{attribute 'GeneratedUsingTerminal: EL6201-0000-0017'}
{attribute addProperty BoxType "EL6201-0000-0017"}
{attribute addProperty Id "Slave_20A_DO0BOOL1Slave_20A_DO1BOOL1Slave_20A_DO2BOOL1Slave_20A_DO3BOOL1Slave_20B_DO0BOOL1Slave_20B_DO1BOOL1Slave_20B_DO2BOOL1Slave_20B_DO3BOOL1"}
{attribute addProperty CRC "2580098861"}
{attribute addProperty Size "8"}
TYPE Slave_20_Outputs_99C92F2D :
STRUCT
	{attribute addProperty Name "Slave_20A_DO0"}
	Slave_20A_DO0 : BOOL;
	{attribute addProperty Name "Slave_20A_DO1"}
	Slave_20A_DO1 : BOOL;
	{attribute addProperty Name "Slave_20A_DO2"}
	Slave_20A_DO2 : BOOL;
	{attribute addProperty Name "Slave_20A_DO3"}
	Slave_20A_DO3 : BOOL;
	{attribute addProperty Name "Slave_20B_DO0"}
	Slave_20B_DO0 : BOOL;
	{attribute addProperty Name "Slave_20B_DO1"}
	Slave_20B_DO1 : BOOL;
	{attribute addProperty Name "Slave_20B_DO2"}
	Slave_20B_DO2 : BOOL;
	{attribute addProperty Name "Slave_20B_DO3"}
	Slave_20B_DO3 : BOOL;
END_STRUCT
END_TYPE

(* stored: Version 1.2.0.0, ProductVersion 3.1.4024.9
   DUT Slave_20_Outputs_99C92F2D: Id {ec432c59-e50f-41c5-9fa6-acdf859f3c59} *)
